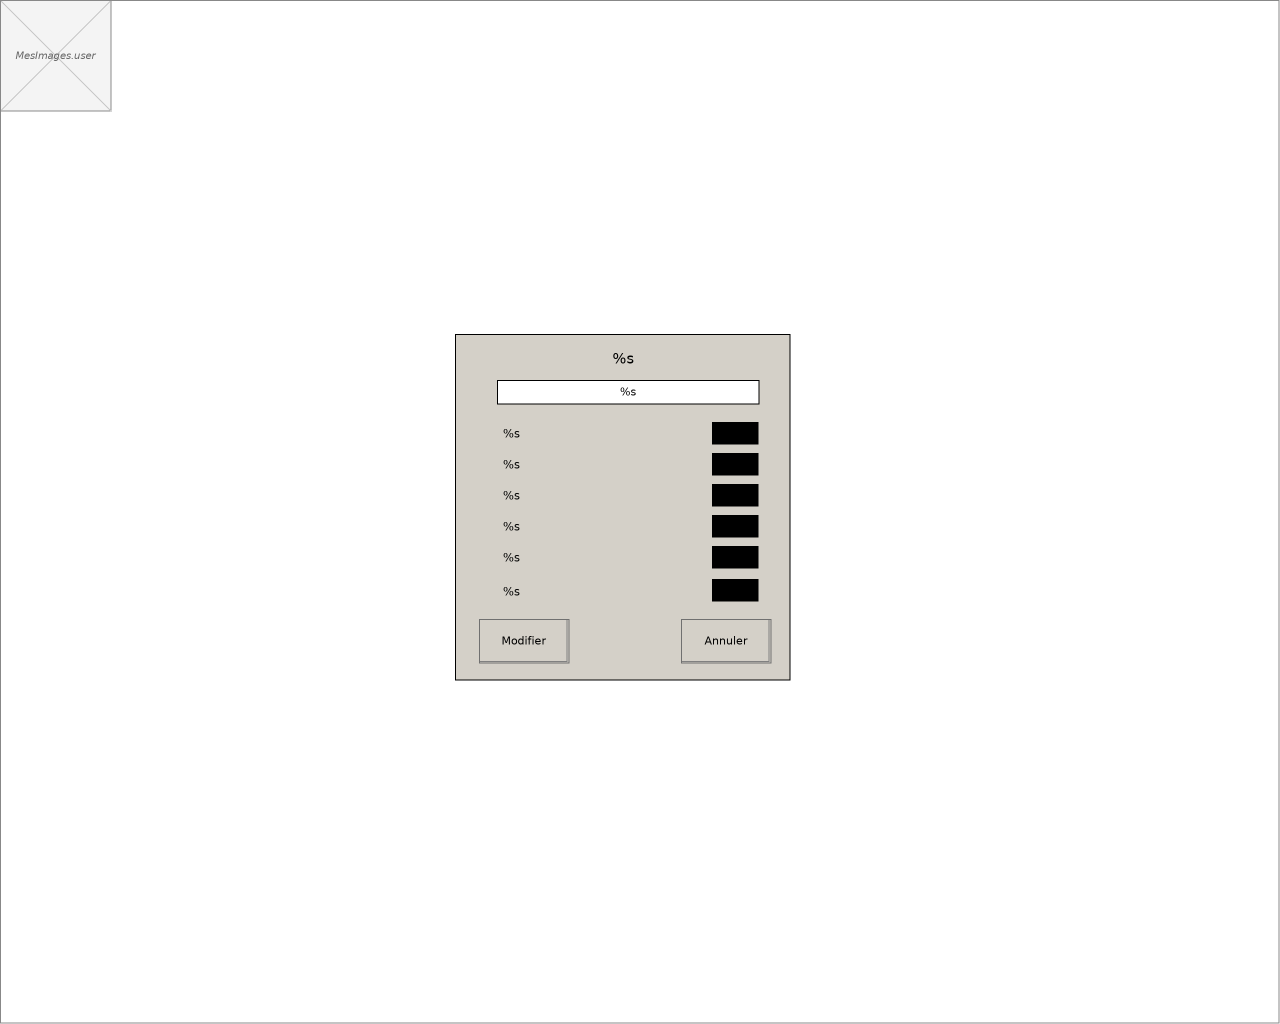
VISUALIZATION UTIL_MOD_GROUP  // 1280x1024
    Image (0,0 111x111), image: MesImages.user
    RoundedRectangle (455,334 335x346)
    Rectangle (460,344 327x29), "%s", text list: 'TextList_Util_Group', text index: 9
    Rectangle (500,450 112x29), "%s", text list: 'TextList_Util_Group', text index: 4
    Rectangle (500,481 112x29), "%s", text list: 'TextList_Util_Group', text index: 5
    Rectangle (500,419 112x29), "%s", text list: 'TextList_Util_Group', text index: 3
    Rectangle (500,512 112x29), "%s", text list: 'TextList_Util_Group', text index: 6
    Rectangle (500,543 112x29), "%s", text list: 'TextList_Util_Group', text index: 7
    Rectangle (500,577 122x29), "%s", text list: 'TextList_Util_Group', text index: 8
    Rectangle (712,422 46x22), "Oui", colour toggle: Global_Variables.PRG_USER.GROUP_TEMP.PROGRAMMATION
        toggle Global_Variables.PRG_USER.GROUP_TEMP.PROGRAMMATION
    Rectangle (712,453 46x22), "Oui", colour toggle: Global_Variables.PRG_USER.GROUP_TEMP.MAINTENANCE
        toggle Global_Variables.PRG_USER.GROUP_TEMP.MAINTENANCE
    Rectangle (712,484 46x22), "Oui", colour toggle: Global_Variables.PRG_USER.GROUP_TEMP.SUPERVISEUR
        toggle Global_Variables.PRG_USER.GROUP_TEMP.SUPERVISEUR
    Rectangle (712,515 46x22), "Oui", colour toggle: Global_Variables.PRG_USER.GROUP_TEMP.PRODUCTION
        toggle Global_Variables.PRG_USER.GROUP_TEMP.PRODUCTION
    Rectangle (712,546 46x22), "Oui", colour toggle: Global_Variables.PRG_USER.GROUP_TEMP.CONF_MACHINE
        toggle Global_Variables.PRG_USER.GROUP_TEMP.CONF_MACHINE
    Rectangle (712,579 46x22), "Oui", colour toggle: Global_Variables.PRG_USER.GROUP_TEMP.FONCTION_SA
        toggle Global_Variables.PRG_USER.GROUP_TEMP.FONCTION_SA
    Button (479,619 90x44), "Modifier", input disabled if: NOT PRG_USER.AUT_NOM_GRP
        toggle PRG_USER.DD_mod_group2
        OnMouseClick: change screen: UTIL_GROUP
    Button (681,619 90x44), "Annuler"
        OnMouseClick: change screen: UTIL_GROUP
    Rectangle (497,380 262x24), "%s", text variable: PRG_USER.GROUP_TEMP.NOM
        OnMouseClick: write the text variable via InputWithLimits
END_VISUALIZATION

(* stored: Version 1.1.0.1, ProductVersion 3.1.4024.10
   Visu UTIL_MOD_GROUP: Id {017c6b36-be02-4800-a056-53f2c77f730d} *)
